PROGRAM GL5A_Accumulation
VAR
	
	RUN_FWD_TO_GL5B_BIT : BOOL; // GL2 EMPTY SO SEND PART FROM GL5 TO GL2
	RUN_FWD_TO_EXIT_BIT : BOOL; // RUN GL5 FWD TO EXIT SENSOR
	
	GL5B_ENTRY_FTRIG:  F_TRIG;
END_VAR
VAR // added by the converter: edge detectors and wires of the graphical bodies
    _w1 : BOOL;
END_VAR

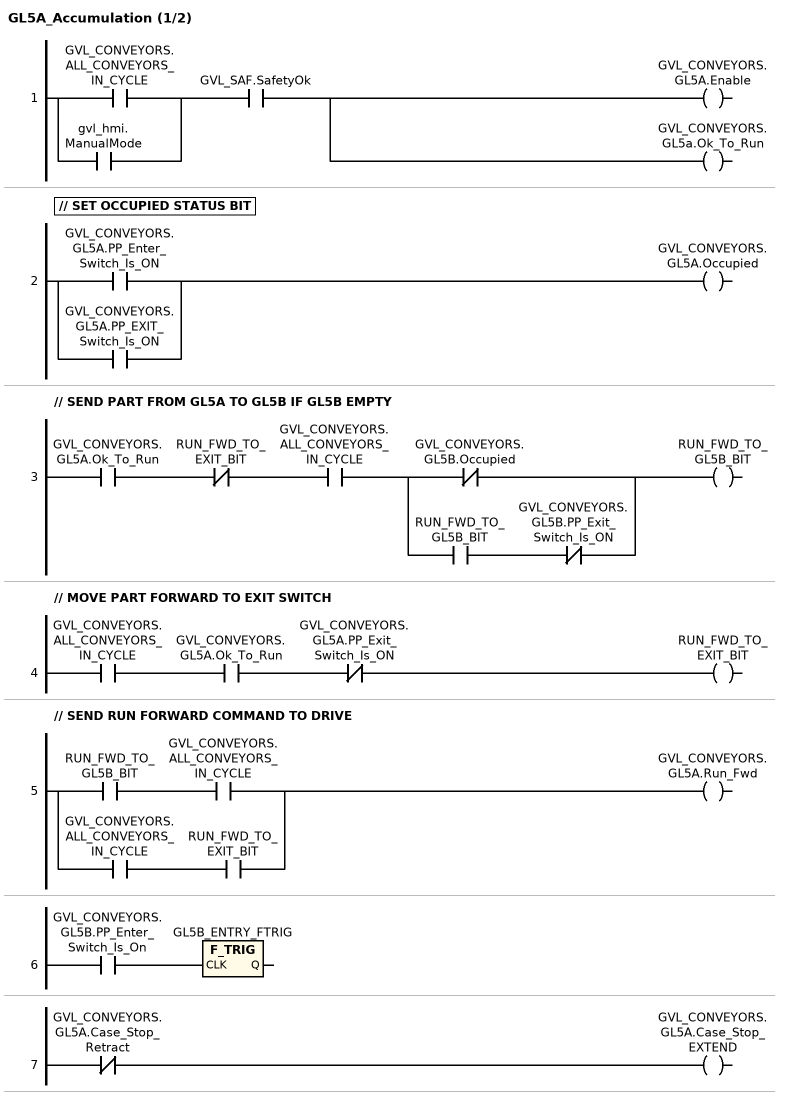
// NETWORK 1
_w1 := (GVL_CONVEYORS.ALL_CONVEYORS_IN_CYCLE OR gvl_hmi.ManualMode) AND GVL_SAF.SafetyOk;
GVL_CONVEYORS.GL5A.Enable := _w1;
GVL_CONVEYORS.GL5a.Ok_To_Run := _w1;

// NETWORK 2
// label: // SET OCCUPIED STATUS BIT
GVL_CONVEYORS.GL5A.Occupied := GVL_CONVEYORS.GL5A.PP_Enter_Switch_Is_ON OR GVL_CONVEYORS.GL5A.PP_EXIT_Switch_Is_ON;

// NETWORK 3: // SEND PART FROM GL5A TO GL5B IF GL5B EMPTY
RUN_FWD_TO_GL5B_BIT := GVL_CONVEYORS.GL5A.Ok_To_Run AND NOT RUN_FWD_TO_EXIT_BIT AND GVL_CONVEYORS.ALL_CONVEYORS_IN_CYCLE AND (NOT GVL_CONVEYORS.GL5B.Occupied OR RUN_FWD_TO_GL5B_BIT AND NOT GVL_CONVEYORS.GL5B.PP_Exit_Switch_Is_ON);

// NETWORK 4: // MOVE PART FORWARD TO EXIT SWITCH
RUN_FWD_TO_EXIT_BIT := GVL_CONVEYORS.ALL_CONVEYORS_IN_CYCLE AND GVL_CONVEYORS.GL5A.Ok_To_Run AND NOT GVL_CONVEYORS.GL5A.PP_Exit_Switch_Is_ON;

// NETWORK 5: // SEND RUN FORWARD COMMAND TO DRIVE
GVL_CONVEYORS.GL5A.Run_Fwd := RUN_FWD_TO_GL5B_BIT AND GVL_CONVEYORS.ALL_CONVEYORS_IN_CYCLE OR GVL_CONVEYORS.ALL_CONVEYORS_IN_CYCLE AND RUN_FWD_TO_EXIT_BIT;

// NETWORK 6
GL5B_ENTRY_FTRIG(CLK := GVL_CONVEYORS.GL5B.PP_Enter_Switch_Is_On); // F_TRIG

// NETWORK 7
GVL_CONVEYORS.GL5A.Case_Stop_EXTEND := NOT GVL_CONVEYORS.GL5A.Case_Stop_Retract;

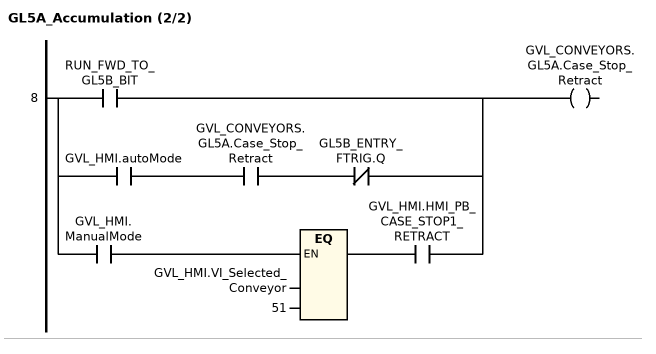
// NETWORK 8
GVL_CONVEYORS.GL5A.Case_Stop_Retract := RUN_FWD_TO_GL5B_BIT OR GVL_HMI.autoMode AND GVL_CONVEYORS.GL5A.Case_Stop_Retract AND NOT GL5B_ENTRY_FTRIG.Q OR (GVL_HMI.ManualMode AND GVL_HMI.VI_Selected_Conveyor = 51) AND GVL_HMI.HMI_PB_CASE_STOP1_RETRACT;

END_PROGRAM

(* stored: Version 1.1.0.1, ProductVersion 3.1.4024.12
   POU GL5A_Accumulation: Id {1b559823-b34b-49ad-8890-b05f77ec0792}, SpecialFunc None *)
